FUNCTION_BLOCK FB_CartSupporLeg EXTENDS FB_CartCtrlBase
VAR_INPUT
END_VAR
VAR_OUTPUT
END_VAR
VAR

	m_actJntPos: Vec8d;
	m_tarJntPos: Vec8d;
	m_initJntPos : Vec8d;
	m_tarJntInc : Vec8d;
	m_maxJntCurrent : ARRAY [1..2] OF LREAL := [800,800];
	m_pinDeployed : ARRAY [1..2] OF BOOL; 
	
	// time threshold to 5-8joint after it's enabled
	m_cartAdjustStartWaitTime :LREAL := 0.2;
	
	//adjust start  time 
	m_adjustStartTime :LREAL;

	m_jntOTG :ARRAY [1..2] OF FB_secOrdTrajFilter;
END_VAR

// override this function in each exact controller
METHOD PROTECTED calcCmdJntPos : BOOL
VAR_IN_OUT CONSTANT
	// slave cart joint data
	i_slaveCart :FB_SlaveCart;
END_VAR

VAR
	i:INT;
END_VAR
//In this method, 8 represents the overhang angle
m_adjustStartTime :=LIMIT(0, m_adjustStartTime + g_cartCtrlCycleTime, 2);
m_actJntPos := i_slaveCart.curJntPos;
IF m_adjustStartTime > m_cartAdjustStartWaitTime THEN
	FOR i:=1 TO 2 DO
		IF ABS(i_slaveCart.curJntCurrent[i]) > m_maxJntCurrent[i] AND ABS(i_slaveCart.curJntVel[i]) < 0.0005 AND m_adjustStartTime >= 2  THEN
			m_pinDeployed[i] := TRUE;
			m_tarJntPos[i] := m_actJntPos[i];
		END_IF
		
		IF FALSE = m_pinDeployed[i] THEN
			m_tarJntPos[i] := m_actJntPos[i] - GVL_CartControlParameters.g_maxJntVel[i] * 2 * g_cartCtrlCycleTime;
		END_IF
		m_jntOTG[i].run(i_targetPos:= m_tarJntPos[i], i_targetVel:= 0.0, o_cmdAcc=> , o_cmdVel=> , o_cmdPos=>m_cmdJntPos[i] );
	END_FOR
	
	IF m_pinDeployed[1] AND m_pinDeployed[2] THEN
		m_isFinished := TRUE;
	END_IF

END_IF
END_METHOD

// override this function in each exact controller
// NOTICE: set joint control mode here, and do some initialization if needed
METHOD PUBLIC init : BOOL
VAR_IN_OUT CONSTANT
	i_slaveCart	:FB_SlaveCart;
END_VAR
VAR_IN_OUT 
	r_cartCtrlCmd :ST_SlaveArmCtrlCmds;
END_VAR
VAR
	i:INT;
END_VAR
//m_holdLastCmds := checkToHoldLastCmds(i_slaveCart);
m_holdLastCmds := checkToHoldLastCmds(i_slaveCart);

SUPER^.init(i_slaveCart,r_cartCtrlCmd);

m_jntEnableFlag[1] :=1;
m_jntEnableFlag[2] :=1;

m_jntOPMode[1]:= DriverOPMode_Pos;
m_jntOPMode[2]:= DriverOPMode_Pos;

m_pinDeployed[1] := FALSE;
m_pinDeployed[2] := FALSE;

m_jntOTG[1].init(i_curCmdPos:= m_cmdJntPos[1], i_curCmdVel:= 0, i_maxV:=GVL_CartControlParameters.g_maxJntVel[1] , i_maxA:=GVL_CartControlParameters.g_maxJntAcc[1] , i_Ts:=g_cartCtrlCycleTime );
m_jntOTG[2].init(i_curCmdPos:= m_cmdJntPos[2], i_curCmdVel:= 0, i_maxV:=GVL_CartControlParameters.g_maxJntVel[2] , i_maxA:=GVL_CartControlParameters.g_maxJntAcc[2] , i_Ts:=g_cartCtrlCycleTime );

m_adjustStartTime := 0;
// update commands to arm
copyCmds(r_cartCtrlCmd);
END_METHOD

END_FUNCTION_BLOCK

(* stored: Version 1.1.0.1, ProductVersion 3.1.4024.11
   POU FB_CartSupporLeg: Id {55d7523f-ccb9-4e03-a220-3c80fe21a70d}, SpecialFunc None
   Method calcCmdJntPos: Id {6b4938eb-71dc-4086-a7ef-b878d82f7a7c}
   Method init: Id {c2bc8804-7c26-45e5-860d-db010c88639a} *)
